// Core §3.8a — DEFAULT station-config provider: in-PLC PERSISTENT records, editable
// locally over OPC UA (§3.10). Remote sources (asset system, MES) substitute later
// through I_StationConfig without touching module code (O1, O6).
FUNCTION_BLOCK FB_LocalStationConfig IMPLEMENTS I_StationConfig
VAR PERSISTENT
    _n : INT;
END_VAR
VAR
    _keys : ARRAY[1..PL_Fraktal.MAX_STATIONCFG] OF STRING(80);
    _ptr  : ARRAY[1..PL_Fraktal.MAX_STATIONCFG] OF PVOID;
    _size : ARRAY[1..PL_Fraktal.MAX_STATIONCFG] OF UDINT;
END_VAR

// no cyclic body

METHOD Load : BOOL
VAR_INPUT
    Key : STRING;
    pCfg : PVOID;
    Size : UDINT;
END_VAR
VAR
    i : INT;
END_VAR
Load := FALSE;
FOR i := 1 TO _n DO
    IF (_keys[i] = Key) AND (_size[i] = Size) AND (pCfg <> 0) THEN
        MEMCPY(destAddr := pCfg, srcAddr := _ptr[i], n := Size);
        Load := TRUE;
        RETURN;
    END_IF
END_FOR
END_METHOD

METHOD Store : BOOL
VAR_INPUT
    Key : STRING;
    pCfg : PVOID;
    Size : UDINT;
END_VAR
VAR
    i : INT;
END_VAR
Store := FALSE;
FOR i := 1 TO _n DO
    IF (_keys[i] = Key) AND (_size[i] = Size) AND (pCfg <> 0) THEN
        MEMCPY(destAddr := _ptr[i], srcAddr := pCfg, n := Size);   // persists (registered targets live in persistent areas)
        Store := TRUE;
        RETURN;
    END_IF
END_FOR
END_METHOD

// application wiring: bind a module's PERSISTENT StationCfg to a key
METHOD Register : BOOL
VAR_INPUT
    Key : STRING(80);
    pData : PVOID;
    Size : UDINT;
END_VAR
IF (_n >= PL_Fraktal.MAX_STATIONCFG) OR (pData = 0) THEN
    Register := FALSE;
    RETURN;
END_IF
_n := _n + 1;
_keys[_n] := Key;
_ptr[_n] := pData;
_size[_n] := Size;
Register := TRUE;
END_METHOD

END_FUNCTION_BLOCK

(* stored: Version 1.1.0.1, ProductVersion 3.1.4024.12
   POU FB_LocalStationConfig: Id {92c257a7-85f6-41e1-96ec-e0f39cbed065}, SpecialFunc None
   Method Load: Id {e1b60d3d-d49d-4e07-8da5-21cf16992a0c}
   Method Store: Id {b310a0c9-7061-4a5d-be51-720b60716df8}
   Method Register: Id {a6063494-7e17-4503-a0ca-6fe0c0f6a8c9} *)
